Staubli VAL3: ClientSend.pgx

public program ClientSend(string x_sMess (dimensions=1))
begin
  sClient=x_sMess
end
